{attribute 'qualified_only'}
VAR_GLOBAL
	
	// Buttons and switches
	bEnableSwitch : BOOL; // ON when either AUTO og MANUAL. OFF when neither. DIGITAL
	bStopSwitch : BOOL;
	bStartSwitch : BOOL;
	bAutoMode : BOOL;
	bManualMode: BOOL;

END_VAR

(* stored: Version 1.1.0.1, ProductVersion 3.1.4024.10
   GVL DigitalInput: Id {d19f44f5-00c3-4ac2-8c88-4611feb238aa} *)
